FUNCTION_BLOCK LogSinkList
VAR_INPUT
END_VAR
VAR_OUTPUT
END_VAR
VAR
	_count		: UINT;
	_iterator			: UINT;
	//~
	_sinks				: ARRAY[0..(MAX_SINKS - 1)] OF ITcoLogSink;
	//~
END_VAR

VAR CONSTANT
	MAX_SINKS				: USINT := 10;
END_VAR

METHOD PUBLIC AddSink : BOOL
VAR_INPUT
	Sink	: ITcoLogSink;
END_VAR
IF _count >= MAX_SINKS - 1 THEN
	AddSink := FALSE;
	RETURN;
END_IF

IF Sink = NULL THEN
	AddSink := FALSE;
	RETURN;
END_IF

_count := _count + 1;
_sinks[_count] := Sink;

AddSink := TRUE;
END_METHOD

METHOD PUBLIC Clear : BOOL
VAR
	i : DINT;
END_VAR
FOR i := 1 TO (MAX_SINKS - 1) DO
	_sinks[i] := NULL;
END_FOR

_count	:= 0;
_iterator		:= 0;
END_METHOD

PROPERTY PUBLIC Count : UINT
GET
Count := _count;
END_GET
END_PROPERTY

METHOD PUBLIC GetNext : ITcoLogSink
VAR_INPUT
END_VAR
_iterator := _iterator + 1;
GetNext := _sinks[_iterator];
END_METHOD

METHOD PUBLIC HasNext : BOOL
VAR_INPUT
END_VAR
IF _iterator < _count THEN
	HasNext := TRUE;
	RETURN;
END_IF

HasNext := FALSE;
END_METHOD

PROPERTY PUBLIC IsEmpty : BOOL
GET
IsEmpty := _count = 0;
END_GET
END_PROPERTY

METHOD PUBLIC ResetIterator : BOOL
VAR_INPUT
END_VAR
_iterator := 0;
END_METHOD

END_FUNCTION_BLOCK

(* stored: Version 1.1.0.1, ProductVersion 3.1.4024.9
   POU LogSinkList: Id {f1dce426-64cb-4330-addf-238cddf067b2}, SpecialFunc None
   Method AddSink: Id {e75037ef-7abc-41b8-a9ba-38adc0f21940}
   Method Clear: Id {f943cee8-a8ab-4d43-b7ad-971195b5660d}
   Property Count: Id {82d97365-6779-4c60-a518-3bc9fcb749be}
   Get Get: Id {accafd36-bfdc-42d3-8904-b3c38d3a0fe3}
   Method GetNext: Id {12452948-f4df-443d-9db8-388982af631a}
   Method HasNext: Id {b896d99e-c897-4507-a057-da4842ed46e8}
   Property IsEmpty: Id {007673dd-60b0-4f31-b0c6-4a57ebce9f35}
   Get Get: Id {6cc4108e-15f7-4e5b-b135-477406524d83}
   Method ResetIterator: Id {0b65297f-6a6b-4ded-b6a7-a95e012a5b69} *)
